// TIA Portal V20 export
VAR_GLOBAL   // PLC tag table "EthernetPortStatus"
END_VAR
VAR_GLOBAL CONSTANT   // user constants
   PN_CPU_X1 : UInt := 0;
   PN_CPU_X2 : UInt := 1;
   PN_RIO : UInt := 2;
   PN_IOLM1 : UInt := 3;
   PN_IOLM2 : UInt := 4;
   PN_IOLM3 : UInt := 5;
   PN_IOLM4 : UInt := 6;
   PN_DRIVE : UInt := 7;
   PN_HMI : UInt := 8;
END_VAR
